(* CoDeSys 2.3 export: CreateBufferHandle.EXP *)

(* POU core/CreateBufferHandle, ST *)
FUNCTION CreateBufferHandle : BOOL
VAR_INPUT
    BufferAddress: DWORD;
    BufferSize: DINT;
END_VAR
VAR_IN_OUT
    Handle: LogBufferHandle;
END_VAR
VAR
    byteOrderInt: INT;
    byteOrderArray: ARRAY[0..1] OF BYTE;
    pInt: POINTER TO INT;
END_VAR
Handle.BufferAddress := BufferAddress;
Handle.BufferSize := BufferSize;
Handle.BufferEndAddress := BufferAddress + (BufferSize - 1);

byteOrderInt := 1;
pInt := ADR(byteOrderArray[0]);
pInt^ := byteOrderInt;
IF byteOrderArray[0] = 1 THEN
    Handle.MagicByte := MAGIC_BYTE_V1_LITTLE_ENDIAN;
ELSE
    Handle.MagicByte := MAGIC_BYTE_V1_BIG_ENDIAN;
END_IF
END_FUNCTION
